SUBAPPLICATION GreenWhiteBackground_Dom (* Subapplication Type *)
  (* Standard: 61499-2 *)
  (* Version 1.0, 2023-02-06, franz *)
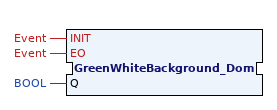
  EVENT_INPUT
    INIT;
    EO;
  END_EVENT
  VAR_INPUT
    Q : BOOL;
  END_VAR
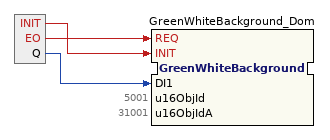
  FBS
    GreenWhiteBackground_Dom : GreenWhiteBackground(u16ObjId := 5001, u16ObjIdA := 31001);
  END_FBS
  EVENT_CONNECTIONS
    EO TO GreenWhiteBackground_Dom.REQ;
    INIT TO GreenWhiteBackground_Dom.INIT;
  END_CONNECTIONS
  DATA_CONNECTIONS
    Q TO GreenWhiteBackground_Dom.DI1;
  END_CONNECTIONS
END_SUBAPPLICATION
